// TIA Portal V19 export
FUNCTION "Assign_Output" : Void   // FC6, LAD
{ S7_Optimized_Access := 'TRUE' }
// stored: SetENOAutomatically false
   VAR_INPUT
      Out : Bool;
      outputSelection : Int;
   END_VAR
   VAR_OUTPUT
      output1 : Bool;
      output2 : Bool;
      output3 : Bool;
      output4 : Bool;
      output5 : Bool;
      output6 : Bool;
      output7 : Bool;
      output8 : Bool;
      output9 : Bool;
      output10 : Bool;
      outputSelected : Int;
   END_VAR
BEGIN

REGION Network 1
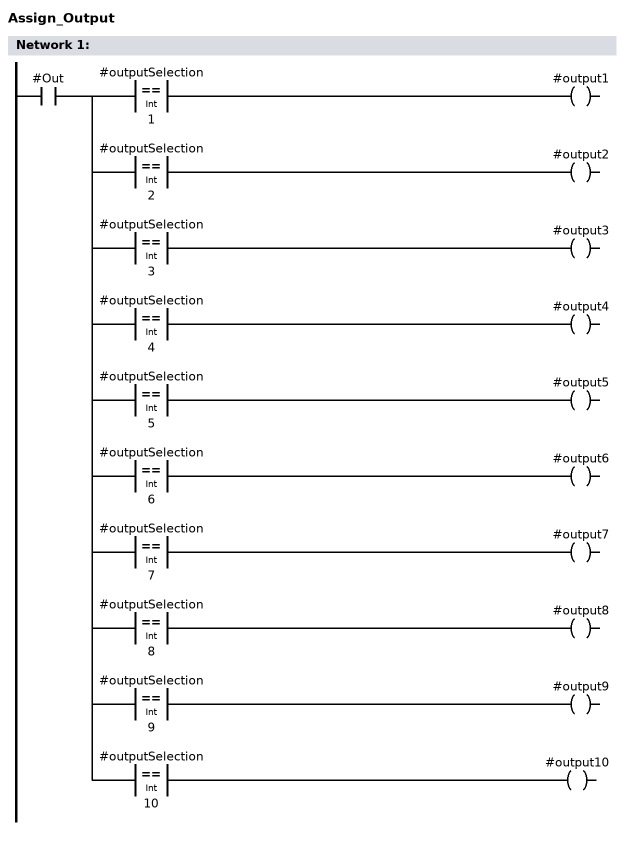
   RUNG wire#powerrail
      Contact( #Out )
      wire#w1
      { S7_Templates := "SrcType := Int" } EQ_Contact(in1 := #outputSelection, in2 := 1)
      Coil( #output1 )
   END_RUNG
   RUNG wire#w1
      { S7_Templates := "SrcType := Int" } EQ_Contact(in1 := #outputSelection, in2 := 2)
      Coil( #output2 )
   END_RUNG
   RUNG wire#w1
      { S7_Templates := "SrcType := Int" } EQ_Contact(in1 := #outputSelection, in2 := 3)
      Coil( #output3 )
   END_RUNG
   RUNG wire#w1
      { S7_Templates := "SrcType := Int" } EQ_Contact(in1 := #outputSelection, in2 := 4)
      Coil( #output4 )
   END_RUNG
   RUNG wire#w1
      { S7_Templates := "SrcType := Int" } EQ_Contact(in1 := #outputSelection, in2 := 5)
      Coil( #output5 )
   END_RUNG
   RUNG wire#w1
      { S7_Templates := "SrcType := Int" } EQ_Contact(in1 := #outputSelection, in2 := 6)
      Coil( #output6 )
   END_RUNG
   RUNG wire#w1
      { S7_Templates := "SrcType := Int" } EQ_Contact(in1 := #outputSelection, in2 := 7)
      Coil( #output7 )
   END_RUNG
   RUNG wire#w1
      { S7_Templates := "SrcType := Int" } EQ_Contact(in1 := #outputSelection, in2 := 8)
      Coil( #output8 )
   END_RUNG
   RUNG wire#w1
      { S7_Templates := "SrcType := Int" } EQ_Contact(in1 := #outputSelection, in2 := 9)
      Coil( #output9 )
   END_RUNG
   RUNG wire#w1
      { S7_Templates := "SrcType := Int" } EQ_Contact(in1 := #outputSelection, in2 := 10)
      Coil( #output10 )
   END_RUNG
   // the same network as SCL:
   #output1 := #Out AND (#outputSelection = 1);
   #output2 := #Out AND (#outputSelection = 2);
   #output3 := #Out AND (#outputSelection = 3);
   #output4 := #Out AND (#outputSelection = 4);
   #output5 := #Out AND (#outputSelection = 5);
   #output6 := #Out AND (#outputSelection = 6);
   #output7 := #Out AND (#outputSelection = 7);
   #output8 := #Out AND (#outputSelection = 8);
   #output9 := #Out AND (#outputSelection = 9);
   #output10 := #Out AND (#outputSelection = 10);
END_REGION
END_FUNCTION
